INTERFACE I_HasCoinState

METHOD PressButton : BOOL
VAR_INPUT
END_VAR
END_METHOD

END_INTERFACE

(* stored: Version 1.1.0.1, ProductVersion 3.1.4022.12
   Itf I_HasCoinState: Id {6657fd82-118c-4979-87e8-20cf36c955eb}
   Method PressButton: Id {a6b076e3-5ac1-4d81-9d74-d4c37a493ba7} *)
